// SIMATIC STEP 7 (V5.x) project PROBLEM 5
// CPU: CPU 314C-2 DP
// station: Hardware
// station: SIMATIC 300(1)
// station: P_ADR_BUS
// program: S7 Program(1)

SYMBOL_TABLE
"1 HZ"	M 0.5	BOOL
"0.5HZ"	M 0.7	BOOL
END_SYMBOL_TABLE

ORGANIZATION_BLOCK OB 1
TITLE = "Main Program Sweep (Cycle)"
//HW8 - PLC - PROBLEM 5
VERSION : 0.1
VAR_TEMP
  OB1_EV_CLASS : BYTE ;	//Bits 0-3 = 1 (Coming event), Bits 4-7 = 1 (Event class 1)
  OB1_SCAN_1 : BYTE ;	//1 (Cold restart scan 1 of OB 1), 3 (Scan 2-n of OB 1)
  OB1_PRIORITY : BYTE ;	//Priority of OB Execution
  OB1_OB_NUMBR : BYTE ;	//1 (Organization block 1, OB1)
  OB1_RESERVED_1 : BYTE ;	//Reserved for system
  OB1_RESERVED_2 : BYTE ;	//Reserved for system
  OB1_PREV_CYCLE : INT ;	//Cycle time of previous OB1 scan (milliseconds)
  OB1_MIN_CYCLE : INT ;	//Minimum cycle time of OB1 (milliseconds)
  OB1_MAX_CYCLE : INT ;	//Maximum cycle time of OB1 (milliseconds)
  OB1_DATE_TIME : DATE_AND_TIME ;	//Date and time OB1 started
END_VAR
BEGIN
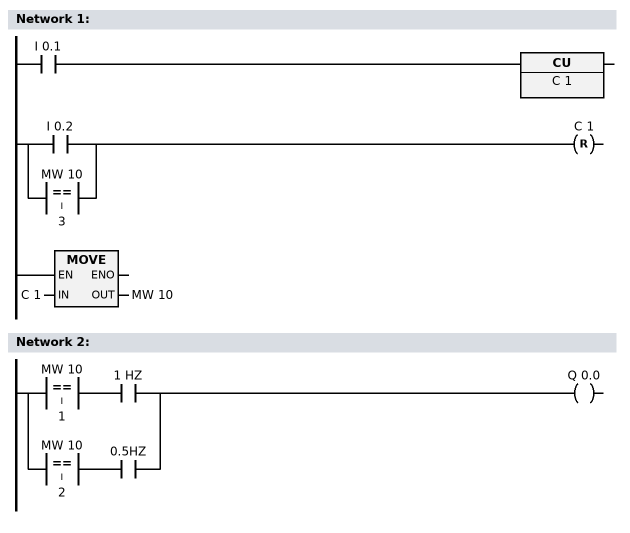
NETWORK
TITLE =
      A     I 0.1;
      CU    C 1;
      BLD   101;
      NOP   0;
      NOP   0;
      A(;
      O     I 0.2;
      O(;
      L     MW 10;
      L     3;
      ==I;
      );
      );
      R     C 1;
      L     C 1;
      T     MW 10;
      NOP   0;
      NOP   0;
NETWORK
TITLE =
      A(;
      L     MW 10;
      L     1;
      ==I;
      );
      A     "1 HZ";
      O;
      A(;
      L     MW 10;
      L     2;
      ==I;
      );
      A     "0.5HZ";
      =     Q 0.0;
END_ORGANIZATION_BLOCK
